(* PLC project SafeLOGIC, BrAutomation SafeDESIGNER  5.24.1.0 *)
(* stored: companyURL http://www.br-automation.com, creationDateTime Sun Dec 07 16:14:24 2025 *)

PROGRAM Main
  VAR  (* added by the conversion: wires and edge detectors of the diagram *)
    _AND_S173_OUT : ANY;
    _OR_S182_OUT : SAFEBOOL;
  END_VAR

(* FBD diagram, written out as Structured Text *)
(* Function 12 - Gas supply interruption *)
_AND_S173_OUT := AND_S(sbSafetyLoop_OK, sDI_Ign_Run, sbN_EngAct_80, sbRel_GV_Purge_OK, sbRel_GV_ERV_PC_OK);
GAS_TRAIN_1(PARA_GT_Exist := SAFETRUE, sbRel_GV := _AND_S173_OUT, bPS_DO_Rel_GVa := bPhysicalState_Rel_GV1a, bPS_DO_Rel_GVb := bPhysicalState_Rel_GV1b, sbGas_LC_Triggered := sbGas_LC_Triggered, sDI_GT_SafeDevOK := sDI_GT1_SafeDevOK, bPS_DO_GT_SafeDev := bPhysicalState_GT1_SafeDev, sbN_Standstill := sbN_Standstill, sbSafetyLoop_OK := sbSafetyLoop_OK, sbSafeInputOK_SafeDevOK := sbSafeInputOK_GT1_SafeDevOK, sbSafeOutputOK_GVa := sbSafeOutputOK_Rel_GV1a, sbSafeOutputOK_GVb := sbSafeOutputOK_Rel_GV1b, sbSafeOutputOK_SafeDev := sbSafeOutputOK_GT1_SafeDev);
bOUT_F12_Rel_GV1 := GAS_TRAIN_1.bOUT_Rel_GV;
sDO_Rel_GV1a := GAS_TRAIN_1.sDO_Rel_GV;
bOUT_F12_Rel_GV1a_PS := GAS_TRAIN_1.bOUT_Rel_GVa_PS;
sDO_Rel_GV1b := GAS_TRAIN_1.sDO_Rel_GV;
bOUT_F12_Rel_GV1b_PS := GAS_TRAIN_1.bOUT_Rel_GVb_PS;
sDO_GT1_SafeDevice := GAS_TRAIN_1.sDO_GT_SafeDevice;
iOUT_F12_GT1_LC_130s_ET := GAS_TRAIN_1.iOUT_GT_LC_130s_ET;
bOUT_F12_GT1_SD_Dem_PS := GAS_TRAIN_1.bOUT_GT_SD_Dem_PS;
bOUT_F12_GT1_SD_Dem := GAS_TRAIN_1.bOUT_GT_SD_Dem;
bAMM_W9528 := GAS_TRAIN_1.bWarning_Out_GVa;
bAMM_W9529 := GAS_TRAIN_1.bWarning_Out_GVb;
bAMM_W9536 := GAS_TRAIN_1.bWarning_In_SafeDevOK;
bAMM_A9421 := GAS_TRAIN_1.bError_GT;
bAMM_W9540 := GAS_TRAIN_1.bWarning_Out_SafeDev;
bOUT_F12_GT1_OK := GAS_TRAIN_1.bOUT_GT_OK;
bOUT_F12_DI_GT1_SafeDevOK := GAS_TRAIN_1.bOUT_DI_GT_SafeDevOK;
GAS_TRAIN_2(PARA_GT_Exist := PARA_GT2_Exist, sbRel_GV := _AND_S173_OUT, bPS_DO_Rel_GVa := bPhysicalState_Rel_GV2a, bPS_DO_Rel_GVb := bPhysicalState_Rel_GV2b, sbGas_LC_Triggered := sbGas_LC_Triggered, sDI_GT_SafeDevOK := sDI_GT2_SafeDevOK, bPS_DO_GT_SafeDev := bPhysicalState_GT2_SafeDev, sbN_Standstill := sbN_Standstill, sbSafetyLoop_OK := sbSafetyLoop_OK, sbSafeInputOK_SafeDevOK := sbSafeInputOK_GT2_SafeDevOK, sbSafeOutputOK_GVa := sbSafeOutputOK_Rel_GV2a, sbSafeOutputOK_GVb := sbSafeOutputOK_Rel_GV2b, sbSafeOutputOK_SafeDev := sbSafeOutputOK_GT2_SafeDev);
bOUT_F12_Rel_GV2 := GAS_TRAIN_2.bOUT_Rel_GV;
sDO_Rel_GV2a := GAS_TRAIN_2.sDO_Rel_GV;
bOUT_F12_Rel_GV2a_PS := GAS_TRAIN_2.bOUT_Rel_GVa_PS;
sDO_Rel_GV2b := GAS_TRAIN_2.sDO_Rel_GV;
bOUT_F12_Rel_GV2b_PS := GAS_TRAIN_2.bOUT_Rel_GVb_PS;
iOUT_F12_GT2_LC_130s_ET := GAS_TRAIN_2.iOUT_GT_LC_130s_ET;
bOUT_F12_GT2_SD_Dem_PS := GAS_TRAIN_2.bOUT_GT_SD_Dem_PS;
sDO_GT2_SafeDevice := GAS_TRAIN_2.sDO_GT_SafeDevice;
bOUT_F12_GT2_SD_Dem := GAS_TRAIN_2.bOUT_GT_SD_Dem;
bAMM_W9530 := GAS_TRAIN_2.bWarning_Out_GVa;
bAMM_W9531 := GAS_TRAIN_2.bWarning_Out_GVb;
bAMM_W9537 := GAS_TRAIN_2.bWarning_In_SafeDevOK;
bAMM_A9422 := GAS_TRAIN_2.bError_GT;
bAMM_W9541 := GAS_TRAIN_2.bWarning_Out_SafeDev;
bOUT_F12_GT2_OK := GAS_TRAIN_2.bOUT_GT_OK;
bOUT_F12_DI_GT2_SafeDevOK := GAS_TRAIN_2.bOUT_DI_GT_SafeDevOK;
GAS_TRAIN_3(PARA_GT_Exist := PARA_GT3_Exist, sbRel_GV := _AND_S173_OUT, bPS_DO_Rel_GVa := bPhysicalState_Rel_GV3a, bPS_DO_Rel_GVb := bPhysicalState_Rel_GV3b, sbGas_LC_Triggered := sbGas_LC_Triggered, sDI_GT_SafeDevOK := sDI_GT3_SafeDevOK, bPS_DO_GT_SafeDev := bPhysicalState_GT3_SafeDev, sbN_Standstill := sbN_Standstill, sbSafetyLoop_OK := sbSafetyLoop_OK, sbSafeInputOK_SafeDevOK := sbSafeInputOK_GT3_SafeDevOK, sbSafeOutputOK_GVa := sbSafeOutputOK_Rel_GV3a, sbSafeOutputOK_GVb := sbSafeOutputOK_Rel_GV3b, sbSafeOutputOK_SafeDev := sbSafeOutputOK_GT3_SafeDev);
bOUT_F12_Rel_GV3 := GAS_TRAIN_3.bOUT_Rel_GV;
sDO_Rel_GV3a := GAS_TRAIN_3.sDO_Rel_GV;
bOUT_F12_Rel_GV3a_PS := GAS_TRAIN_3.bOUT_Rel_GVa_PS;
sDO_Rel_GV3b := GAS_TRAIN_3.sDO_Rel_GV;
bOUT_F12_Rel_GV3b_PS := GAS_TRAIN_3.bOUT_Rel_GVb_PS;
sDO_GT3_SafeDevice := GAS_TRAIN_3.sDO_GT_SafeDevice;
bAMM_W9532 := GAS_TRAIN_3.bWarning_Out_GVa;
bAMM_W9533 := GAS_TRAIN_3.bWarning_Out_GVb;
bAMM_W9538 := GAS_TRAIN_3.bWarning_In_SafeDevOK;
iOUT_F12_GT3_LC_130s_ET := GAS_TRAIN_3.iOUT_GT_LC_130s_ET;
bAMM_A9423 := GAS_TRAIN_3.bError_GT;
bOUT_F12_GT3_SD_Dem_PS := GAS_TRAIN_3.bOUT_GT_SD_Dem_PS;
bOUT_F12_GT3_SD_Dem := GAS_TRAIN_3.bOUT_GT_SD_Dem;
bAMM_W9542 := GAS_TRAIN_3.bWarning_Out_SafeDev;
bOUT_F12_GT3_OK := GAS_TRAIN_3.bOUT_GT_OK;
bOUT_F12_DI_GT3_SafeDevOK := GAS_TRAIN_3.bOUT_DI_GT_SafeDevOK;
GAS_TRAIN_4(PARA_GT_Exist := PARA_GT4_Exist, sbRel_GV := _AND_S173_OUT, bPS_DO_Rel_GVa := bPhysicalState_Rel_GV4a, bPS_DO_Rel_GVb := bPhysicalState_Rel_GV4b, sbGas_LC_Triggered := sbGas_LC_Triggered, sDI_GT_SafeDevOK := sDI_GT4_SafeDevOK, bPS_DO_GT_SafeDev := bPhysicalState_GT4_SafeDev, sbN_Standstill := sbN_Standstill, sbSafetyLoop_OK := sbSafetyLoop_OK, sbSafeInputOK_SafeDevOK := sbSafeInputOK_GT4_SafeDevOK, sbSafeOutputOK_GVa := sbSafeOutputOK_Rel_GV4a, sbSafeOutputOK_GVb := sbSafeOutputOK_Rel_GV4b, sbSafeOutputOK_SafeDev := sbSafeOutputOK_GT4_SafeDev);
bOUT_F12_Rel_GV4 := GAS_TRAIN_4.bOUT_Rel_GV;
sDO_Rel_GV4a := GAS_TRAIN_4.sDO_Rel_GV;
bOUT_F12_Rel_GV4a_PS := GAS_TRAIN_4.bOUT_Rel_GVa_PS;
sDO_Rel_GV4b := GAS_TRAIN_4.sDO_Rel_GV;
bOUT_F12_Rel_GV4b_PS := GAS_TRAIN_4.bOUT_Rel_GVb_PS;
sDO_GT4_SafeDevice := GAS_TRAIN_4.sDO_GT_SafeDevice;
iOUT_F12_GT4_LC_130s_ET := GAS_TRAIN_4.iOUT_GT_LC_130s_ET;
bOUT_F12_GT4_SD_Dem_PS := GAS_TRAIN_4.bOUT_GT_SD_Dem_PS;
bOUT_F12_GT4_SD_Dem := GAS_TRAIN_4.bOUT_GT_SD_Dem;
bAMM_W9534 := GAS_TRAIN_4.bWarning_Out_GVa;
bAMM_W9535 := GAS_TRAIN_4.bWarning_Out_GVb;
bAMM_W9539 := GAS_TRAIN_4.bWarning_In_SafeDevOK;
bAMM_A9424 := GAS_TRAIN_4.bError_GT;
bAMM_W9543 := GAS_TRAIN_4.bWarning_Out_SafeDev;
bOUT_F12_GT4_OK := GAS_TRAIN_4.bOUT_GT_OK;
bOUT_F12_DI_GT4_SafeDevOK := GAS_TRAIN_4.bOUT_DI_GT_SafeDevOK;
GAS_TRAIN_DCGA(PARA_GT_Exist := PARA_DCGA_Exist, sbRel_GV := _AND_S173_OUT, bPS_DO_Rel_GVa := bPhysicalState_Rel_GVa_DCGA, bPS_DO_Rel_GVb := bPhysicalState_Rel_GVb_DCGA, sbGas_LC_Triggered := sbGas_LC_Triggered, sDI_GT_SafeDevOK := sDI_DCGA_SafeDevOK, bPS_DO_GT_SafeDev := bPhysicalState_DCGA_SafeDev, sbN_Standstill := sbN_Standstill, sbSafetyLoop_OK := sbSafetyLoop_OK, sbSafeInputOK_SafeDevOK := sbSafeInputOK_DCGA_SafeDevOK, sbSafeOutputOK_GVa := sbSafeOutputOK_Rel_GVa_DCGA, sbSafeOutputOK_GVb := sbSafeOutputOK_Rel_GVb_DCGA, sbSafeOutputOK_SafeDev := sbSafeOutputOK_DCGA_SafeDev);
bOUT_F12_Rel_GV_DCGA := GAS_TRAIN_DCGA.bOUT_Rel_GV;
sDO_Rel_GVa_DCGA := GAS_TRAIN_DCGA.sDO_Rel_GV;
bOUT_F12_Rel_GVa_DCGA_PS := GAS_TRAIN_DCGA.bOUT_Rel_GVa_PS;
sDO_Rel_GVb_DCGA := GAS_TRAIN_DCGA.sDO_Rel_GV;
bOUT_F12_Rel_GVb_DCGA_PS := GAS_TRAIN_DCGA.bOUT_Rel_GVb_PS;
iOUT_F12_DCGA_LC_130s_ET := GAS_TRAIN_DCGA.iOUT_GT_LC_130s_ET;
bOUT_F12_DCGA_SD_Dem_PS := GAS_TRAIN_DCGA.bOUT_GT_SD_Dem_PS;
sDO_DCGA_SafeDevice := GAS_TRAIN_DCGA.sDO_GT_SafeDevice;
bOUT_F12_DCGA_SD_Dem := GAS_TRAIN_DCGA.bOUT_GT_SD_Dem;
bAMM_W9701 := GAS_TRAIN_DCGA.bWarning_Out_GVa;
bAMM_W9702 := GAS_TRAIN_DCGA.bWarning_Out_GVb;
bAMM_W9703 := GAS_TRAIN_DCGA.bWarning_In_SafeDevOK;
bAMM_A9484 := GAS_TRAIN_DCGA.bError_GT;
bAMM_W9704 := GAS_TRAIN_DCGA.bWarning_Out_SafeDev;
bOUT_F12_DCGA_OK := GAS_TRAIN_DCGA.bOUT_GT_OK;
bOUT_F12_DI_DCGA_SafeDevOK := GAS_TRAIN_DCGA.bOUT_DI_GT_SafeDevOK;
xR_TRIG_F12_LC(CLK := sbN_EngOperation);
xF_TRIG_F12_LC(CLK := sDO_GT1_SafeDevice);
xRS_F12_LC(SET := xR_TRIG_F12_LC.Q, RESET1 := xF_TRIG_F12_LC.Q);
sbGas_LC_Triggered := xRS_F12_LC.Q1;
(* Physical state *)
(* Gas valves opened *)
_OR_S182_OUT := OR_S(BOOL_TO_SAFEBOOL(bPhysicalState_Rel_GV1a), BOOL_TO_SAFEBOOL(bPhysicalState_Rel_GV1b), BOOL_TO_SAFEBOOL(bPhysicalState_Rel_GV2a), BOOL_TO_SAFEBOOL(bPhysicalState_Rel_GV2b), BOOL_TO_SAFEBOOL(bPhysicalState_Rel_GV3a), BOOL_TO_SAFEBOOL(bPhysicalState_Rel_GV3b), BOOL_TO_SAFEBOOL(bPhysicalState_Rel_GV4a), BOOL_TO_SAFEBOOL(bPhysicalState_Rel_GV4b), BOOL_TO_SAFEBOOL(bPhysicalState_Rel_GVa_DCGA), BOOL_TO_SAFEBOOL(bPhysicalState_Rel_GVb_DCGA));
sbGasValves_Open := _OR_S182_OUT;
sbGasValves_Closed := NOT_S(_OR_S182_OUT);
(* Gas valves opened for 1s *)
xTON_F12_GasV_Open_1s(IN := _OR_S182_OUT, PT := SAFETIME#1s);
sbGasValves_Open_1s := xTON_F12_GasV_Open_1s.Q;
(* Gas valves opened for 10s *)
xTON_F12_GasV_Open_10s(IN := _OR_S182_OUT, PT := SAFETIME#10s);
sbGasValves_Open_10s := xTON_F12_GasV_Open_10s.Q;
(* Gas valves opened for 60s *)
(* Elapsed time *)
xET_GV_Open_60s(IN := sbGasValves_Open, PT := SAFETIME#60s);
iOUT_F12_GV_Open_60s_ET := xET_GV_Open_60s.iOUT_ET;
sbGasValves_Open_60s := xET_GV_Open_60s.Q;
(* Safety loop *)
(* Safety loop *)
sbF12_OK_Gas := AND_S(AND_S(BOOL_TO_SAFEBOOL(bAMM_A9421), BOOL_TO_SAFEBOOL(bAMM_A9422), BOOL_TO_SAFEBOOL(bAMM_A9423), BOOL_TO_SAFEBOOL(bAMM_A9424), BOOL_TO_SAFEBOOL(bAMM_A9484), BOOL_TO_SAFEBOOL(bAMM_W9701), BOOL_TO_SAFEBOOL(bAMM_W9702), BOOL_TO_SAFEBOOL(bAMM_W9703), BOOL_TO_SAFEBOOL(bAMM_W9704)), AND_S(BOOL_TO_SAFEBOOL(bAMM_W9528), BOOL_TO_SAFEBOOL(bAMM_W9529), BOOL_TO_SAFEBOOL(bAMM_W9530), BOOL_TO_SAFEBOOL(bAMM_W9531), BOOL_TO_SAFEBOOL(bAMM_W9532), BOOL_TO_SAFEBOOL(bAMM_W9533), BOOL_TO_SAFEBOOL(bAMM_W9534), BOOL_TO_SAFEBOOL(bAMM_W9535), BOOL_TO_SAFEBOOL(bAMM_W9536), BOOL_TO_SAFEBOOL(bAMM_W9537), BOOL_TO_SAFEBOOL(bAMM_W9538), BOOL_TO_SAFEBOOL(bAMM_W9539), BOOL_TO_SAFEBOOL(bAMM_W9540), BOOL_TO_SAFEBOOL(bAMM_W9541), BOOL_TO_SAFEBOOL(bAMM_W9542), BOOL_TO_SAFEBOOL(bAMM_W9543)));
END_PROGRAM
